(*udt (user defined type) of Beckhoff EP3174_0002 - 4 channel,  Analog Input Terminal:*)


TYPE udt_EP3174_0002 :
STRUCT

	CH1: INT;
	CH2: INT;
	CH3: INT;
	CH4: INT;
	InfoData: udt_ECATSlave_Status;

END_STRUCT
END_TYPE

(* stored: Version 1.1.0.1, ProductVersion 3.1.4024.9
   DUT udt_EP3174_0002: Id {b074afea-ec01-4bcb-ae6d-3e1ae947838d} *)
